TYPE
    TcoUrRobotics_T2O_TCP_IO :
    STRUCT
        bArray AT %I* : ARRAY[0..75] OF BYTE;
    END_STRUCT
END_TYPE

(* stored: Version 1.1.0.1, ProductVersion 3.1.4024.12
   DUT TcoUrRobotics_T2O_TCP_IO: Id {9e10f247-7e22-0ce2-2674-2415f4de9bb5} *)
